# EPICS substitutions: iocBoot/ioc13test/asynRecord.substitutions
file "$(ASYN)/db/asynRecord.db"
{
pattern
{P              R         PORT     ADDR  OMAX IMAX}
{13TEST:     serial1   serial1    0    256  256}
{13TEST:     serial2   serial2    0    256  256}
}
